{attribute 'GeneratedUsingTerminal: KL9900-0059'}
{attribute addProperty BoxType "KL9900-0059"}
{attribute addProperty Description ""}
{attribute addProperty Physics ""}
{attribute addProperty Id "Channel_1AT %Q*Channel_707BD1FE0"}
{attribute addProperty CRC "3686840388"}
{attribute addProperty Size "0"}
TYPE KL_DBC0B844 :
STRUCT
	{attribute addProperty Name "Channel_1"}
	Channel_1 : Channel_707BD1FE;
END_STRUCT
END_TYPE

(* stored: Version 1.2.0.0, ProductVersion 3.1.4024.11
   DUT KL_DBC0B844: Id {1d4dadf0-14eb-4ad9-8628-eac9f5800017} *)
